// Implicitly generated code : DO NOT EDIT
FUNCTION CheckRangeUnsigned : UDINT
VAR_INPUT
	value, lower, upper: UDINT;
END_VAR

// Implicitly generated code : Only an Implementation suggestion
IF (value < lower) THEN
	CheckRangeUnsigned := lower;
	GVL_Checks.dCheckRangeUnsigned := GVL_Checks.dCheckRangeUnsigned + 1;
ELSIF(value > upper) THEN
	CheckRangeUnsigned := upper;
	GVL_Checks.dCheckRangeUnsigned := GVL_Checks.dCheckRangeUnsigned + 1;
ELSE
	CheckRangeUnsigned := value;
END_IF

END_FUNCTION

(* stored: Version 1.1.0.1, ProductVersion 3.1.4020.3
   POU CheckRangeUnsigned: Id {36bf99f8-15d6-410e-b338-663fb75109d2}, SpecialFunc CheckRangeUnsigned *)
